// TIA Portal V19 export
FUNCTION "Posisjonering" : Void   // FC2, LAD
{ S7_Optimized_Access := 'TRUE' }
// stored: SetENOAutomatically false
BEGIN

REGION Network 1
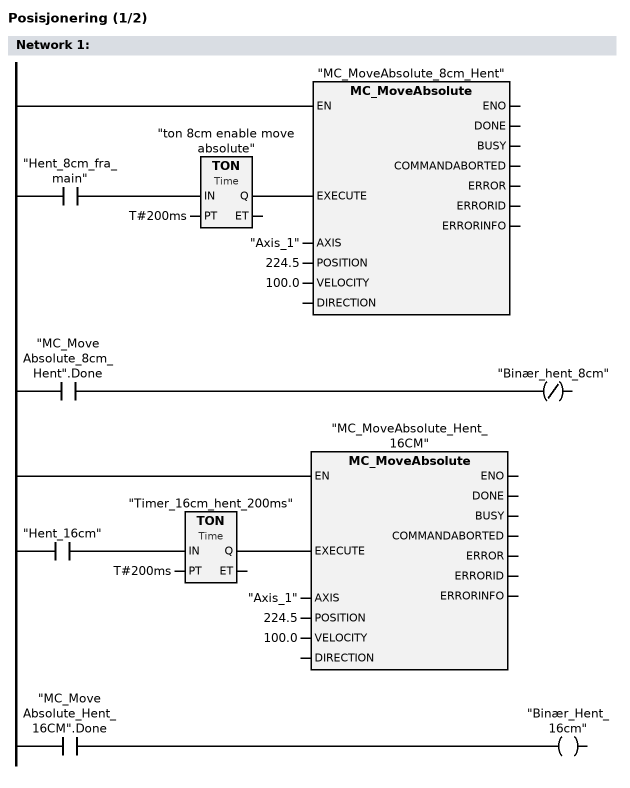
   RUNG wire#powerrail
      "MC_MoveAbsolute_8cm_Hent".MC_MoveAbsolute(Execute := wire#w1, Axis := "Axis_1", Position := 224.5, Velocity := 100.0, Direction :=, Done =>, Busy =>, CommandAborted =>, Error =>, ErrorID =>, ErrorInfo =>)
   END_RUNG
   RUNG wire#powerrail
      Contact( "Hent_8cm_fra_main" )
      { S7_Templates := "time_type := Time" } "ton 8cm enable move absolute".TON(pt := T#200ms, et =>)
   END_RUNG wire#w1
   RUNG wire#powerrail
      Contact( "MC_MoveAbsolute_8cm_Hent".Done )
      I_Coil( "Binær_hent_8cm" )
   END_RUNG
   RUNG wire#powerrail
      "MC_MoveAbsolute_Hent_16CM".MC_MoveAbsolute(Execute := wire#w2, Axis := "Axis_1", Position := 224.5, Velocity := 100.0, Direction :=, Done =>, Busy =>, CommandAborted =>, Error =>, ErrorID =>, ErrorInfo =>)
   END_RUNG
   RUNG wire#powerrail
      Contact( "Hent_16cm" )
      { S7_Templates := "time_type := Time" } "Timer_16cm_hent_200ms".TON(pt := T#200ms, et =>)
   END_RUNG wire#w2
   RUNG wire#powerrail
      Contact( "MC_MoveAbsolute_Hent_16CM".Done )
      Coil( "Binær_Hent_16cm" )
   END_RUNG
   // the same network as SCL:
   "ton 8cm enable move absolute".TON(IN := "Hent_8cm_fra_main", PT := T#200ms);
   "MC_MoveAbsolute_8cm_Hent"(Execute := "ton 8cm enable move absolute".Q,   // MC_MoveAbsolute
                           Axis := "Axis_1",
                           Position := 224.5,
                           Velocity := 100.0);
   "Binær_hent_8cm" := NOT "MC_MoveAbsolute_8cm_Hent".Done;
   "Timer_16cm_hent_200ms".TON(IN := "Hent_16cm", PT := T#200ms);
   "MC_MoveAbsolute_Hent_16CM"(Execute := "Timer_16cm_hent_200ms".Q,   // MC_MoveAbsolute
                           Axis := "Axis_1",
                           Position := 224.5,
                           Velocity := 100.0);
   "Binær_Hent_16cm" := "MC_MoveAbsolute_Hent_16CM".Done;
END_REGION

REGION Network 2
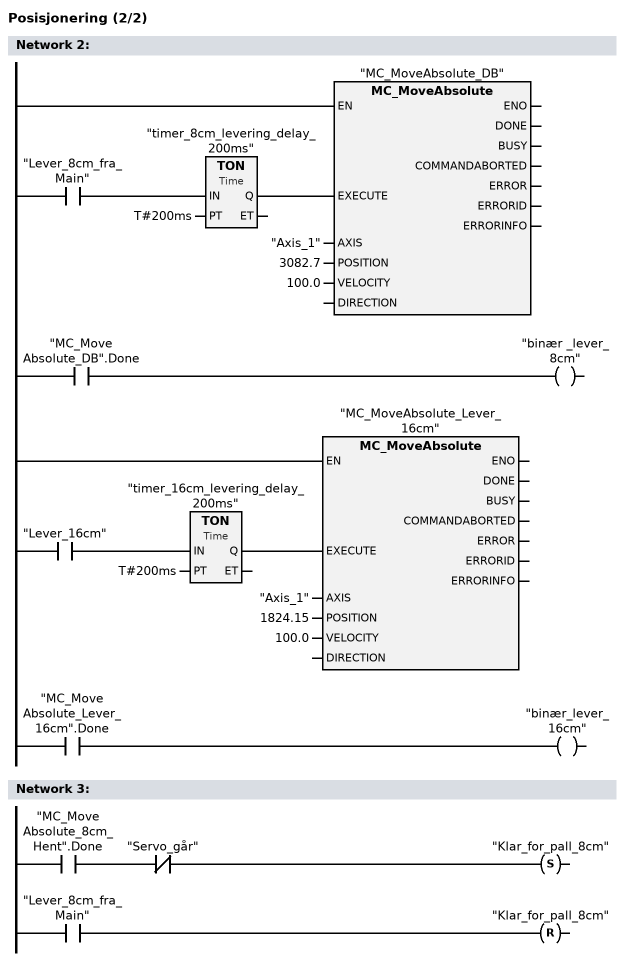
   RUNG wire#powerrail
      "MC_MoveAbsolute_DB".MC_MoveAbsolute(Execute := wire#w1, Axis := "Axis_1", Position := 3082.7, Velocity := 100.0, Direction :=, Done =>, Busy =>, CommandAborted =>, Error =>, ErrorID =>, ErrorInfo =>)
   END_RUNG
   RUNG wire#powerrail
      Contact( "Lever_8cm_fra_Main" )
      { S7_Templates := "time_type := Time" } "timer_8cm_levering_delay_200ms".TON(pt := T#200ms, et =>)
   END_RUNG wire#w1
   RUNG wire#powerrail
      Contact( "MC_MoveAbsolute_DB".Done )
      Coil( "binær _lever_8cm" )
   END_RUNG
   RUNG wire#powerrail
      "MC_MoveAbsolute_Lever_16cm".MC_MoveAbsolute(Execute := wire#w2, Axis := "Axis_1", Position := 1824.15, Velocity := 100.0, Direction :=, Done =>, Busy =>, CommandAborted =>, Error =>, ErrorID =>, ErrorInfo =>)
   END_RUNG
   RUNG wire#powerrail
      Contact( "Lever_16cm" )
      { S7_Templates := "time_type := Time" } "timer_16cm_levering_delay_200ms".TON(pt := T#200ms, et =>)
   END_RUNG wire#w2
   RUNG wire#powerrail
      Contact( "MC_MoveAbsolute_Lever_16cm".Done )
      Coil( "binær_lever_16cm" )
   END_RUNG
   // the same network as SCL:
   "timer_8cm_levering_delay_200ms".TON(IN := "Lever_8cm_fra_Main", PT := T#200ms);
   "MC_MoveAbsolute_DB"(Execute := "timer_8cm_levering_delay_200ms".Q,   // MC_MoveAbsolute
                        Axis := "Axis_1",
                        Position := 3082.7,
                        Velocity := 100.0);
   "binær _lever_8cm" := "MC_MoveAbsolute_DB".Done;
   "timer_16cm_levering_delay_200ms".TON(IN := "Lever_16cm", PT := T#200ms);
   "MC_MoveAbsolute_Lever_16cm"(Execute := "timer_16cm_levering_delay_200ms".Q,   // MC_MoveAbsolute
                           Axis := "Axis_1",
                           Position := 1824.15,
                           Velocity := 100.0);
   "binær_lever_16cm" := "MC_MoveAbsolute_Lever_16cm".Done;
END_REGION

REGION Network 3
   RUNG wire#powerrail
      Contact( "MC_MoveAbsolute_8cm_Hent".Done )
      I_Contact( "Servo_går" )
      S_Coil( "Klar_for_pall_8cm" )
   END_RUNG
   RUNG wire#powerrail
      Contact( "Lever_8cm_fra_Main" )
      R_Coil( "Klar_for_pall_8cm" )
   END_RUNG
   // the same network as SCL:
   IF "MC_MoveAbsolute_8cm_Hent".Done AND NOT "Servo_går" THEN "Klar_for_pall_8cm" := TRUE; END_IF;
   IF "Lever_8cm_fra_Main" THEN "Klar_for_pall_8cm" := FALSE; END_IF;
END_REGION
END_FUNCTION
